// TIA Portal V18 export
DATA_BLOCK "settings"   // DB12
{ S7_Optimized_Access := 'TRUE' }
// stored: InstanceOfName UDT_settings, InstanceOfType UDT
"UDT_settings"
   // VAR RETAIN
   //    taktTimeCntOption { ExternalVisible := 'False'; S7_SetPoint := 'True'} : DInt;
   //    target { ExternalVisible := 'False'; S7_SetPoint := 'True'} : DInt;
   //    taktTime { ExternalVisible := 'False'; S7_SetPoint := 'True'} : DInt;
   //    countOption { ExternalVisible := 'False'; S7_SetPoint := 'True'} : DInt;
   // END_VAR
BEGIN
END_DATA_BLOCK
